(* IEC 61131-3 sources: Std_PalletMover/Class/SpeedCalculator, 1 file *)

(* ---- SpeedCalculator.st ---- *)
(*!
<Class
	Name               = "SpeedCalculator"
	Revision           = "0.0"
	RealtimeTask       = "false"
	CyclicTask         = "true"
	BackgroundTask     = "false"
	Sigmatek           = "false"
	OSInterface        = "false"
	HighPriority       = "false"
	Automatic          = "false"
	UpdateMode         = "Prescan"
	SharedCommandTable = "true"
	Objectsize         = "(810,120)">
	<Channels>
		<Server Name="ClassSvr" Visualized="false" Initialize="false" WriteProtected="true" Retentive="false"/>
		<Server Name="mms" Visualized="false" Initialize="false" WriteProtected="true" Retentive="false"/>
		<Client Name="SafetyPulsjes" Required="false" Internal="false"/>
	</Channels>
</Class>
*)
SpeedCalculator : CLASS
  //Servers:
	ClassSvr 	: SvrChCmd_DINT;
	mms 	: SvrCh_REAL;
  //Clients:
	SafetyPulsjes 	: CltCh_DINT;
  //Variables:
		_OldPulses 	: DINT;
  //Functions:

	FUNCTION VIRTUAL GLOBAL CyWork
		VAR_INPUT
			EAX 	: UDINT;
		END_VAR
		VAR_OUTPUT
			state (EAX) 	: UDINT := READY;
		END_VAR;
  //Tables:
	FUNCTION @STD
		VAR_OUTPUT
			ret_code	: CONFSTATES;
		END_VAR;
	FUNCTION GLOBAL TAB @CT_;
END_CLASS;

FUNCTION VIRTUAL GLOBAL SpeedCalculator::CyWork
	VAR_INPUT
		EAX 	: UDINT;
	END_VAR
	VAR_OUTPUT
		state (EAX) 	: UDINT;(* := READY *)
	END_VAR
  VAR
  	DiffPulsjes : dint;
    Rondjes : real;
  END_VAR

  SafetyPulsjes := SafetyPulsjes.Read();

  DiffPulsjes := SafetyPulsjes - _OldPulses;
  if DiffPulsjes <> 0 then
    Rondjes := to_real(DiffPulsjes) / 1024.0;
    mms := Rondjes / 57.76 / 1.5 * 973.8937;
  end_if;

  _OldPulses := SafetyPulsjes;

END_FUNCTION
